// TIA Portal V20 export
FUNCTION "FNet_Map07" : Void   // FC143, LAD
// stored: Namespace CITI_Logic, SetENOAutomatically false
   VAR_TEMP
      FlexNet_DataString_PUN : Array[1..20] of Char;
      FlexNet_GM_PartNumber : Array[1..8] of Char;
      FlexNet_OptionalData : Array[1..12] of Char;
      FlexNet_Tracking_ID1 : Array[1..32] of Char;
      FlexNet_Track_ID1_Attrib : Array[1..20] of Char;
      FlexNet_Tracking_ID2 : Array[1..32] of Char;
      FlexNet_Track_ID2_Attrib : Array[1..20] of Char;
      FlexNet_Tracking_ID3 : Array[1..32] of Char;
      FlexNet_Track_ID3_Attrib : Array[1..20] of Char;
      FlexNet_Tracking_ID4 : Array[1..32] of Char;
      FlexNet_Track_ID4_Attrib : Array[1..20] of Char;
      FlexNet_Tracking_ID5 : Array[1..32] of Char;
      FlexNet_Track_ID5_Attrib : Array[1..20] of Char;
      FlexNet_Tracking_ID6 : Array[1..32] of Char;
      FlexNet_Track_ID6_Attrib : Array[1..20] of Char;
      FlexNet_Tracking_ID7 : Array[1..32] of Char;
      FlexNet_Track_ID7_Attrib : Array[1..20] of Char;
      FlexNet_Tracking_ID8 : Array[1..32] of Char;
      FlexNet_Track_ID8_Attrib : Array[1..20] of Char;
      FlexNet_Tracking_ID9 : Array[1..32] of Char;
      FlexNet_Track_ID9_Attrib : Array[1..20] of Char;
      FlexNet_Tracking_ID10 : Array[1..32] of Char;
      FlexNet_Track_ID10_Attrib : Array[1..20] of Char;
      TEMP_OEM_FnetNoRespWarn : Bool;   // REPLACE THIS WITH CORRECT WARNING BIT
      TEMP_OEM_FnetRetryOccur : Bool;   // REPLACE THIS WITH CORRECT WARNING BIT
      TEMP_OEM_FN_NoResponseL2 : Byte;
      OEM_FN_DATA_RECVD : Bool;
      TracePoint : Bool;
      Marriage : Bool;
      QualityGate : Bool;
      HostQuery : Bool;
      OEM_to_Populate_FN_RESPONSE_COUNTS_ALLOWED : Int;
   END_VAR
   VAR_TEMP   // added for the SCL form of the ladder/FBD networks
      _w1 : Bool;
      _w2 : Bool;
   END_VAR
BEGIN

REGION Network 1: Part Pass
   // **Replace the "CITI_Logic_Setup".OEM_TO_COMPLETE Bit with the correct Logic to drive the signal**
   // 
   // Set the Pass Bit Always True for a Trace Point, Marriage, and Host Query.
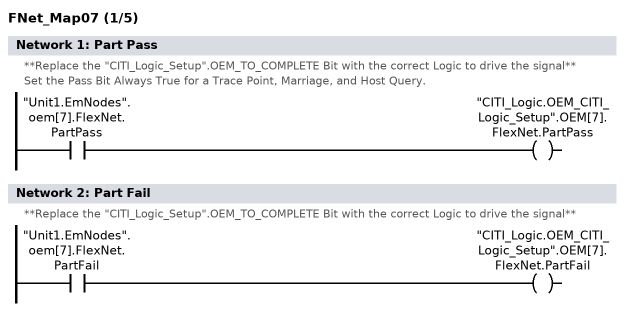
   RUNG wire#powerrail
      Contact( "Unit1.EmNodes".oem[7].FlexNet.PartPass )
      Coil( "CITI_Logic.OEM_CITI_Logic_Setup".OEM[7].FlexNet.PartPass )
   END_RUNG
   // the same network as SCL:
   "CITI_Logic.OEM_CITI_Logic_Setup".OEM[7].FlexNet.PartPass := "Unit1.EmNodes".oem[7].FlexNet.PartPass;
END_REGION

REGION Network 2: Part Fail
   // **Replace the "CITI_Logic_Setup".OEM_TO_COMPLETE Bit with the correct Logic to drive the signal**
   RUNG wire#powerrail
      Contact( "Unit1.EmNodes".oem[7].FlexNet.PartFail )
      Coil( "CITI_Logic.OEM_CITI_Logic_Setup".OEM[7].FlexNet.PartFail )
   END_RUNG
   // the same network as SCL:
   "CITI_Logic.OEM_CITI_Logic_Setup".OEM[7].FlexNet.PartFail := "Unit1.EmNodes".oem[7].FlexNet.PartFail;
END_REGION

REGION Network 3: Pun, GM Part Number, Optional Data, Tracking ID, Tracking ID Attribute, and Data Ready
   // **Replace the "CITI_Logic_Setup".OEM_TO_COMPLETE Bit with the correct Logic to drive the signal**
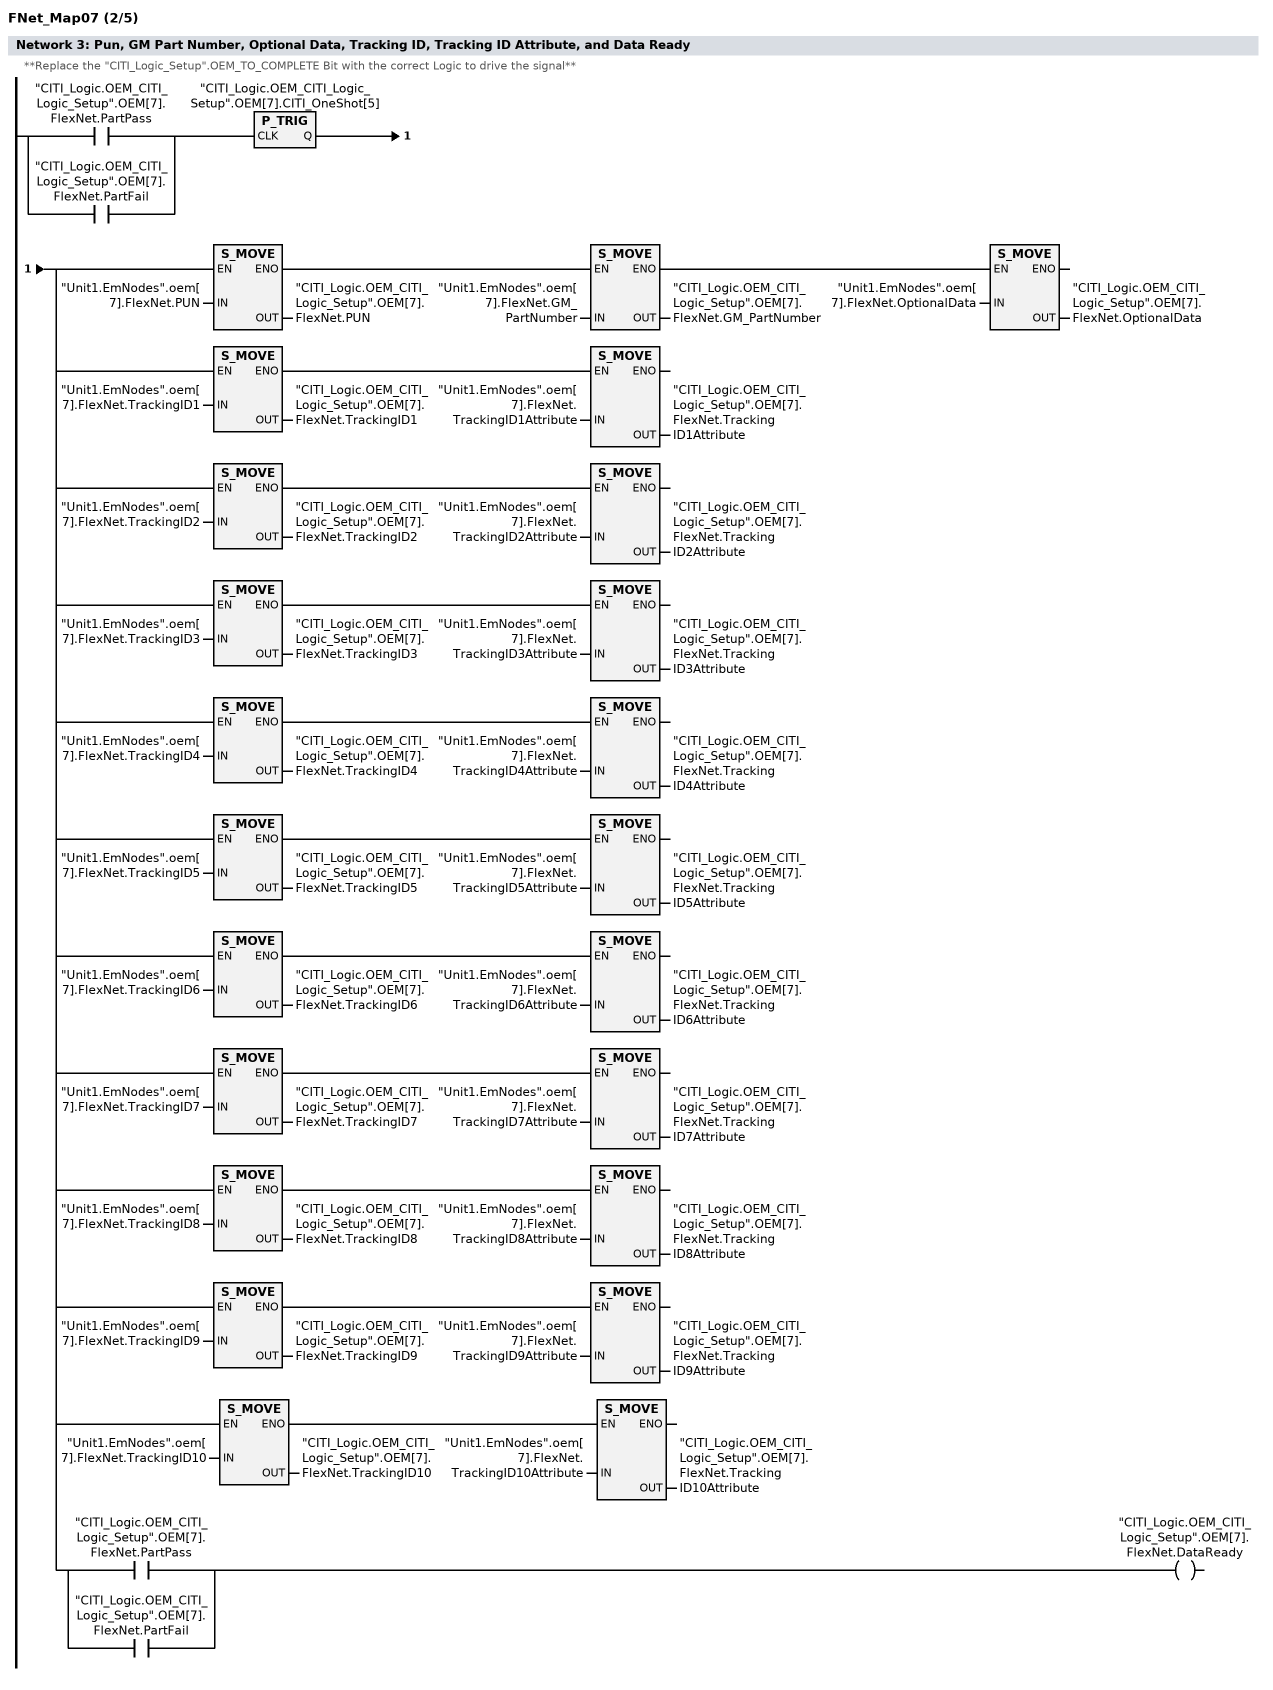
   RUNG wire#powerrail
      Contact( "CITI_Logic.OEM_CITI_Logic_Setup".OEM[7].FlexNet.PartPass )
      wire#w1
      P_Trig( "CITI_Logic.OEM_CITI_Logic_Setup".OEM[7].CITI_OneShot[5] )
      wire#w2
      S_Move(in := "Unit1.EmNodes".oem[7].FlexNet.PUN, out => "CITI_Logic.OEM_CITI_Logic_Setup".OEM[7].FlexNet.PUN)
      S_Move(in := "Unit1.EmNodes".oem[7].FlexNet.GM_PartNumber, out => "CITI_Logic.OEM_CITI_Logic_Setup".OEM[7].FlexNet.GM_PartNumber)
      S_Move(in := "Unit1.EmNodes".oem[7].FlexNet.OptionalData, out => "CITI_Logic.OEM_CITI_Logic_Setup".OEM[7].FlexNet.OptionalData)
   END_RUNG
   RUNG wire#powerrail
      Contact( "CITI_Logic.OEM_CITI_Logic_Setup".OEM[7].FlexNet.PartFail )
   END_RUNG wire#w1
   RUNG wire#w2
      S_Move(in := "Unit1.EmNodes".oem[7].FlexNet.TrackingID1, out => "CITI_Logic.OEM_CITI_Logic_Setup".OEM[7].FlexNet.TrackingID1)
      S_Move(in := "Unit1.EmNodes".oem[7].FlexNet.TrackingID1Attribute, out => "CITI_Logic.OEM_CITI_Logic_Setup".OEM[7].FlexNet.TrackingID1Attribute)
   END_RUNG
   RUNG wire#w2
      S_Move(in := "Unit1.EmNodes".oem[7].FlexNet.TrackingID2, out => "CITI_Logic.OEM_CITI_Logic_Setup".OEM[7].FlexNet.TrackingID2)
      S_Move(in := "Unit1.EmNodes".oem[7].FlexNet.TrackingID2Attribute, out => "CITI_Logic.OEM_CITI_Logic_Setup".OEM[7].FlexNet.TrackingID2Attribute)
   END_RUNG
   RUNG wire#w2
      S_Move(in := "Unit1.EmNodes".oem[7].FlexNet.TrackingID3, out => "CITI_Logic.OEM_CITI_Logic_Setup".OEM[7].FlexNet.TrackingID3)
      S_Move(in := "Unit1.EmNodes".oem[7].FlexNet.TrackingID3Attribute, out => "CITI_Logic.OEM_CITI_Logic_Setup".OEM[7].FlexNet.TrackingID3Attribute)
   END_RUNG
   RUNG wire#w2
      S_Move(in := "Unit1.EmNodes".oem[7].FlexNet.TrackingID4, out => "CITI_Logic.OEM_CITI_Logic_Setup".OEM[7].FlexNet.TrackingID4)
      S_Move(in := "Unit1.EmNodes".oem[7].FlexNet.TrackingID4Attribute, out => "CITI_Logic.OEM_CITI_Logic_Setup".OEM[7].FlexNet.TrackingID4Attribute)
   END_RUNG
   RUNG wire#w2
      S_Move(in := "Unit1.EmNodes".oem[7].FlexNet.TrackingID5, out => "CITI_Logic.OEM_CITI_Logic_Setup".OEM[7].FlexNet.TrackingID5)
      S_Move(in := "Unit1.EmNodes".oem[7].FlexNet.TrackingID5Attribute, out => "CITI_Logic.OEM_CITI_Logic_Setup".OEM[7].FlexNet.TrackingID5Attribute)
   END_RUNG
   RUNG wire#w2
      S_Move(in := "Unit1.EmNodes".oem[7].FlexNet.TrackingID6, out => "CITI_Logic.OEM_CITI_Logic_Setup".OEM[7].FlexNet.TrackingID6)
      S_Move(in := "Unit1.EmNodes".oem[7].FlexNet.TrackingID6Attribute, out => "CITI_Logic.OEM_CITI_Logic_Setup".OEM[7].FlexNet.TrackingID6Attribute)
   END_RUNG
   RUNG wire#w2
      S_Move(in := "Unit1.EmNodes".oem[7].FlexNet.TrackingID7, out => "CITI_Logic.OEM_CITI_Logic_Setup".OEM[7].FlexNet.TrackingID7)
      S_Move(in := "Unit1.EmNodes".oem[7].FlexNet.TrackingID7Attribute, out => "CITI_Logic.OEM_CITI_Logic_Setup".OEM[7].FlexNet.TrackingID7Attribute)
   END_RUNG
   RUNG wire#w2
      S_Move(in := "Unit1.EmNodes".oem[7].FlexNet.TrackingID8, out => "CITI_Logic.OEM_CITI_Logic_Setup".OEM[7].FlexNet.TrackingID8)
      S_Move(in := "Unit1.EmNodes".oem[7].FlexNet.TrackingID8Attribute, out => "CITI_Logic.OEM_CITI_Logic_Setup".OEM[7].FlexNet.TrackingID8Attribute)
   END_RUNG
   RUNG wire#w2
      S_Move(in := "Unit1.EmNodes".oem[7].FlexNet.TrackingID9, out => "CITI_Logic.OEM_CITI_Logic_Setup".OEM[7].FlexNet.TrackingID9)
      S_Move(in := "Unit1.EmNodes".oem[7].FlexNet.TrackingID9Attribute, out => "CITI_Logic.OEM_CITI_Logic_Setup".OEM[7].FlexNet.TrackingID9Attribute)
   END_RUNG
   RUNG wire#w2
      S_Move(in := "Unit1.EmNodes".oem[7].FlexNet.TrackingID10, out => "CITI_Logic.OEM_CITI_Logic_Setup".OEM[7].FlexNet.TrackingID10)
      S_Move(in := "Unit1.EmNodes".oem[7].FlexNet.TrackingID10Attribute, out => "CITI_Logic.OEM_CITI_Logic_Setup".OEM[7].FlexNet.TrackingID10Attribute)
   END_RUNG
   RUNG wire#w2
      Contact( "CITI_Logic.OEM_CITI_Logic_Setup".OEM[7].FlexNet.PartPass )
      wire#w3
      Coil( "CITI_Logic.OEM_CITI_Logic_Setup".OEM[7].FlexNet.DataReady )
   END_RUNG
   RUNG wire#w2
      Contact( "CITI_Logic.OEM_CITI_Logic_Setup".OEM[7].FlexNet.PartFail )
   END_RUNG wire#w3
   // the same network as SCL:
   #_w1 := "CITI_Logic.OEM_CITI_Logic_Setup".OEM[7].FlexNet.PartPass OR "CITI_Logic.OEM_CITI_Logic_Setup".OEM[7].FlexNet.PartFail;
   #_w2 := #_w1 AND NOT "CITI_Logic.OEM_CITI_Logic_Setup".OEM[7].CITI_OneShot[5];   // rising edge
   "CITI_Logic.OEM_CITI_Logic_Setup".OEM[7].CITI_OneShot[5] := #_w1;
   IF #_w2 THEN
       "CITI_Logic.OEM_CITI_Logic_Setup".OEM[7].FlexNet.PUN := "Unit1.EmNodes".oem[7].FlexNet.PUN;
       "CITI_Logic.OEM_CITI_Logic_Setup".OEM[7].FlexNet.GM_PartNumber := "Unit1.EmNodes".oem[7].FlexNet.GM_PartNumber;
       "CITI_Logic.OEM_CITI_Logic_Setup".OEM[7].FlexNet.OptionalData := "Unit1.EmNodes".oem[7].FlexNet.OptionalData;
       "CITI_Logic.OEM_CITI_Logic_Setup".OEM[7].FlexNet.TrackingID1 := "Unit1.EmNodes".oem[7].FlexNet.TrackingID1;
       "CITI_Logic.OEM_CITI_Logic_Setup".OEM[7].FlexNet.TrackingID1Attribute := "Unit1.EmNodes".oem[7].FlexNet.TrackingID1Attribute;
       "CITI_Logic.OEM_CITI_Logic_Setup".OEM[7].FlexNet.TrackingID2 := "Unit1.EmNodes".oem[7].FlexNet.TrackingID2;
       "CITI_Logic.OEM_CITI_Logic_Setup".OEM[7].FlexNet.TrackingID2Attribute := "Unit1.EmNodes".oem[7].FlexNet.TrackingID2Attribute;
       "CITI_Logic.OEM_CITI_Logic_Setup".OEM[7].FlexNet.TrackingID3 := "Unit1.EmNodes".oem[7].FlexNet.TrackingID3;
       "CITI_Logic.OEM_CITI_Logic_Setup".OEM[7].FlexNet.TrackingID3Attribute := "Unit1.EmNodes".oem[7].FlexNet.TrackingID3Attribute;
       "CITI_Logic.OEM_CITI_Logic_Setup".OEM[7].FlexNet.TrackingID4 := "Unit1.EmNodes".oem[7].FlexNet.TrackingID4;
       "CITI_Logic.OEM_CITI_Logic_Setup".OEM[7].FlexNet.TrackingID4Attribute := "Unit1.EmNodes".oem[7].FlexNet.TrackingID4Attribute;
       "CITI_Logic.OEM_CITI_Logic_Setup".OEM[7].FlexNet.TrackingID5 := "Unit1.EmNodes".oem[7].FlexNet.TrackingID5;
       "CITI_Logic.OEM_CITI_Logic_Setup".OEM[7].FlexNet.TrackingID5Attribute := "Unit1.EmNodes".oem[7].FlexNet.TrackingID5Attribute;
       "CITI_Logic.OEM_CITI_Logic_Setup".OEM[7].FlexNet.TrackingID6 := "Unit1.EmNodes".oem[7].FlexNet.TrackingID6;
       "CITI_Logic.OEM_CITI_Logic_Setup".OEM[7].FlexNet.TrackingID6Attribute := "Unit1.EmNodes".oem[7].FlexNet.TrackingID6Attribute;
       "CITI_Logic.OEM_CITI_Logic_Setup".OEM[7].FlexNet.TrackingID7 := "Unit1.EmNodes".oem[7].FlexNet.TrackingID7;
       "CITI_Logic.OEM_CITI_Logic_Setup".OEM[7].FlexNet.TrackingID7Attribute := "Unit1.EmNodes".oem[7].FlexNet.TrackingID7Attribute;
       "CITI_Logic.OEM_CITI_Logic_Setup".OEM[7].FlexNet.TrackingID8 := "Unit1.EmNodes".oem[7].FlexNet.TrackingID8;
       "CITI_Logic.OEM_CITI_Logic_Setup".OEM[7].FlexNet.TrackingID8Attribute := "Unit1.EmNodes".oem[7].FlexNet.TrackingID8Attribute;
       "CITI_Logic.OEM_CITI_Logic_Setup".OEM[7].FlexNet.TrackingID9 := "Unit1.EmNodes".oem[7].FlexNet.TrackingID9;
       "CITI_Logic.OEM_CITI_Logic_Setup".OEM[7].FlexNet.TrackingID9Attribute := "Unit1.EmNodes".oem[7].FlexNet.TrackingID9Attribute;
       "CITI_Logic.OEM_CITI_Logic_Setup".OEM[7].FlexNet.TrackingID10 := "Unit1.EmNodes".oem[7].FlexNet.TrackingID10;
       "CITI_Logic.OEM_CITI_Logic_Setup".OEM[7].FlexNet.TrackingID10Attribute := "Unit1.EmNodes".oem[7].FlexNet.TrackingID10Attribute;
   END_IF;
   "CITI_Logic.OEM_CITI_Logic_Setup".OEM[7].FlexNet.DataReady := #_w2 AND ("CITI_Logic.OEM_CITI_Logic_Setup".OEM[7].FlexNet.PartPass OR "CITI_Logic.OEM_CITI_Logic_Setup".OEM[7].FlexNet.PartFail);
END_REGION

REGION Network 4: Transaction Type
   // **Replace the "CITI_Logic_Setup".OEM_TO_COMPLETE Bit with the correct Logic to drive the signal**
   // 
   // For the Transaction Type:
   //  
   // Flexnet TypeInteger Value
   // Trace Point = 1
   // Marriage = 2
   // Quality Gate = 4
   // Host Query = 8
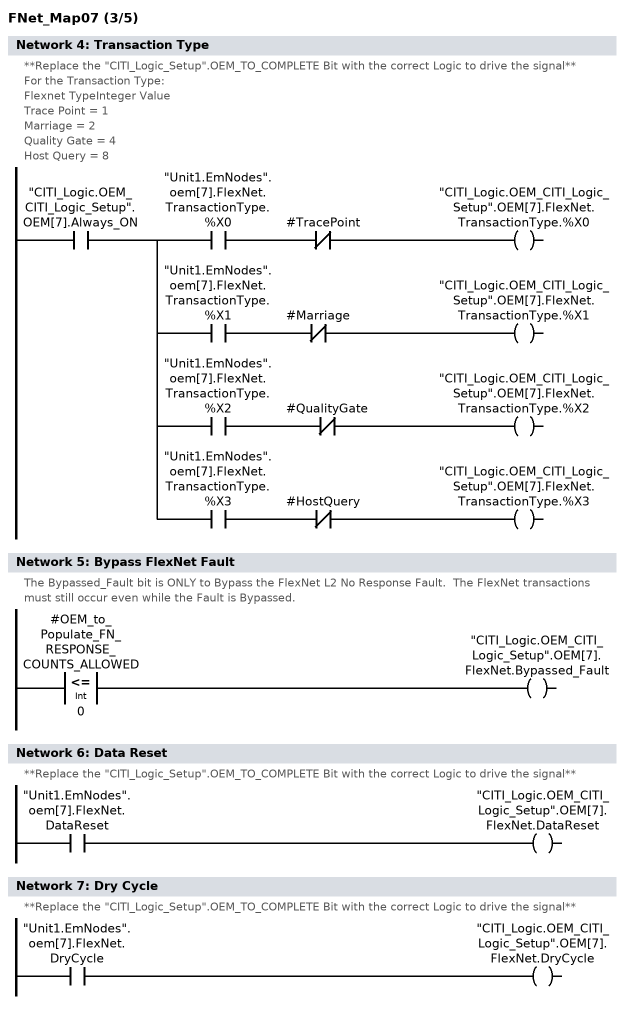
   RUNG wire#powerrail
      Contact( "CITI_Logic.OEM_CITI_Logic_Setup".OEM[7].Always_ON )
      wire#w1
      Contact( "Unit1.EmNodes".oem[7].FlexNet.TransactionType.%X0 )
      I_Contact( #TracePoint )
      Coil( "CITI_Logic.OEM_CITI_Logic_Setup".OEM[7].FlexNet.TransactionType.%X0 )
   END_RUNG
   RUNG wire#w1
      Contact( "Unit1.EmNodes".oem[7].FlexNet.TransactionType.%X1 )
      I_Contact( #Marriage )
      Coil( "CITI_Logic.OEM_CITI_Logic_Setup".OEM[7].FlexNet.TransactionType.%X1 )
   END_RUNG
   RUNG wire#w1
      Contact( "Unit1.EmNodes".oem[7].FlexNet.TransactionType.%X2 )
      I_Contact( #QualityGate )
      Coil( "CITI_Logic.OEM_CITI_Logic_Setup".OEM[7].FlexNet.TransactionType.%X2 )
   END_RUNG
   RUNG wire#w1
      Contact( "Unit1.EmNodes".oem[7].FlexNet.TransactionType.%X3 )
      I_Contact( #HostQuery )
      Coil( "CITI_Logic.OEM_CITI_Logic_Setup".OEM[7].FlexNet.TransactionType.%X3 )
   END_RUNG
   // the same network as SCL:
   #_w1 := "CITI_Logic.OEM_CITI_Logic_Setup".OEM[7].Always_ON;
   "CITI_Logic.OEM_CITI_Logic_Setup".OEM[7].FlexNet.TransactionType.%X0 := "CITI_Logic.OEM_CITI_Logic_Setup".OEM[7].Always_ON AND "Unit1.EmNodes".oem[7].FlexNet.TransactionType.%X0 AND NOT #TracePoint;
   "CITI_Logic.OEM_CITI_Logic_Setup".OEM[7].FlexNet.TransactionType.%X1 := #_w1 AND "Unit1.EmNodes".oem[7].FlexNet.TransactionType.%X1 AND NOT #Marriage;
   "CITI_Logic.OEM_CITI_Logic_Setup".OEM[7].FlexNet.TransactionType.%X2 := #_w1 AND "Unit1.EmNodes".oem[7].FlexNet.TransactionType.%X2 AND NOT #QualityGate;
   "CITI_Logic.OEM_CITI_Logic_Setup".OEM[7].FlexNet.TransactionType.%X3 := #_w1 AND "Unit1.EmNodes".oem[7].FlexNet.TransactionType.%X3 AND NOT #HostQuery;
END_REGION

REGION Network 5: Bypass FlexNet Fault
   // The Bypassed_Fault bit is ONLY to Bypass the FlexNet L2 No Response Fault.  The FlexNet transactions must still occur even while the Fault is Bypassed.
   RUNG wire#powerrail
      { S7_Templates := "SrcType := Int" } LE_Contact(in1 := #OEM_to_Populate_FN_RESPONSE_COUNTS_ALLOWED, in2 := 0)
      Coil( "CITI_Logic.OEM_CITI_Logic_Setup".OEM[7].FlexNet.Bypassed_Fault )
   END_RUNG
   // the same network as SCL:
   "CITI_Logic.OEM_CITI_Logic_Setup".OEM[7].FlexNet.Bypassed_Fault := #OEM_to_Populate_FN_RESPONSE_COUNTS_ALLOWED <= 0;
END_REGION

REGION Network 6: Data Reset
   // **Replace the "CITI_Logic_Setup".OEM_TO_COMPLETE Bit with the correct Logic to drive the signal**
   RUNG wire#powerrail
      Contact( "Unit1.EmNodes".oem[7].FlexNet.DataReset )
      Coil( "CITI_Logic.OEM_CITI_Logic_Setup".OEM[7].FlexNet.DataReset )
   END_RUNG
   // the same network as SCL:
   "CITI_Logic.OEM_CITI_Logic_Setup".OEM[7].FlexNet.DataReset := "Unit1.EmNodes".oem[7].FlexNet.DataReset;
END_REGION

REGION Network 7: Dry Cycle
   // **Replace the "CITI_Logic_Setup".OEM_TO_COMPLETE Bit with the correct Logic to drive the signal**
   RUNG wire#powerrail
      Contact( "Unit1.EmNodes".oem[7].FlexNet.DryCycle )
      Coil( "CITI_Logic.OEM_CITI_Logic_Setup".OEM[7].FlexNet.DryCycle )
   END_RUNG
   // the same network as SCL:
   "CITI_Logic.OEM_CITI_Logic_Setup".OEM[7].FlexNet.DryCycle := "Unit1.EmNodes".oem[7].FlexNet.DryCycle;
END_REGION

REGION Network 8: FlexNet 10 Child Block Call
   // Input time for response fault can be directly entered or from another source.
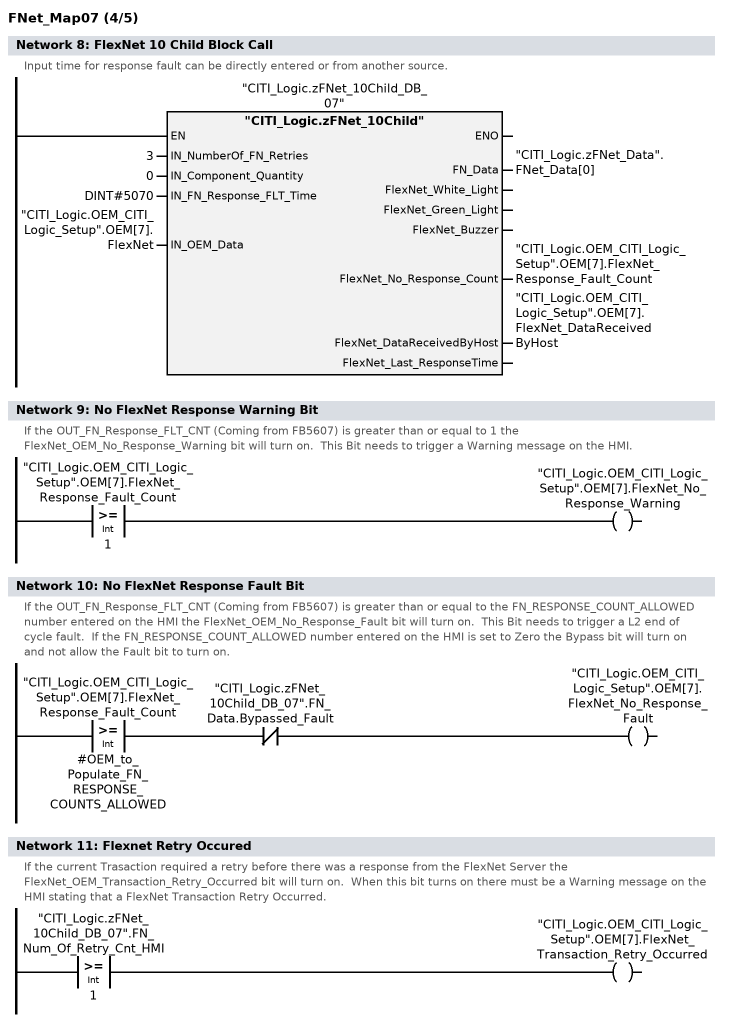
   RUNG wire#powerrail
      "CITI_Logic.zFNet_10Child_DB_07"(IN_NumberOf_FN_Retries := 3, IN_Component_Quantity := 0, IN_FN_Response_FLT_Time := DINT#5070, IN_OEM_Data := "CITI_Logic.OEM_CITI_Logic_Setup".OEM[7].FlexNet, FN_Data => "CITI_Logic.zFNet_Data".FNet_Data[0], FlexNet_White_Light =>, FlexNet_Green_Light =>, FlexNet_Buzzer =>, FlexNet_No_Response_Count => "CITI_Logic.OEM_CITI_Logic_Setup".OEM[7].FlexNet_Response_Fault_Count, FlexNet_DataReceivedByHost => "CITI_Logic.OEM_CITI_Logic_Setup".OEM[7].FlexNet_DataReceivedByHost, FlexNet_Last_ResponseTime =>)
   END_RUNG
   // the same network as SCL:
   "CITI_Logic.zFNet_10Child_DB_07"(IN_NumberOf_FN_Retries := 3,   // "CITI_Logic.zFNet_10Child"
                           IN_Component_Quantity := 0,
                           IN_FN_Response_FLT_Time := DINT#5070,
                           IN_OEM_Data := "CITI_Logic.OEM_CITI_Logic_Setup".OEM[7].FlexNet,
                           FN_Data => "CITI_Logic.zFNet_Data".FNet_Data[0],
                           FlexNet_No_Response_Count => "CITI_Logic.OEM_CITI_Logic_Setup".OEM[7].FlexNet_Response_Fault_Count,
                           FlexNet_DataReceivedByHost => "CITI_Logic.OEM_CITI_Logic_Setup".OEM[7].FlexNet_DataReceivedByHost);
END_REGION

REGION Network 9: No FlexNet Response Warning Bit
   // If the OUT_FN_Response_FLT_CNT (Coming from FB5607) is greater than or equal to 1 the FlexNet_OEM_No_Response_Warning bit will turn on.  This Bit needs to trigger a Warning message on the HMI.
   RUNG wire#powerrail
      { S7_Templates := "SrcType := Int" } GE_Contact(in1 := "CITI_Logic.OEM_CITI_Logic_Setup".OEM[7].FlexNet_Response_Fault_Count, in2 := 1)
      Coil( "CITI_Logic.OEM_CITI_Logic_Setup".OEM[7].FlexNet_No_Response_Warning )
   END_RUNG
   // the same network as SCL:
   "CITI_Logic.OEM_CITI_Logic_Setup".OEM[7].FlexNet_No_Response_Warning := "CITI_Logic.OEM_CITI_Logic_Setup".OEM[7].FlexNet_Response_Fault_Count >= 1;
END_REGION

REGION Network 10: No FlexNet Response Fault Bit
   // If the OUT_FN_Response_FLT_CNT (Coming from FB5607) is greater than or equal to the FN_RESPONSE_COUNT_ALLOWED number entered on the HMI the FlexNet_OEM_No_Response_Fault bit will turn on.  This Bit needs to trigger a L2 end of cycle fault.  If the FN_RESPONSE_COUNT_ALLOWED number entered on the HMI is set to Zero the Bypass bit will turn on and not allow the Fault bit to turn on.
   RUNG wire#powerrail
      { S7_Templates := "SrcType := Int" } GE_Contact(in1 := "CITI_Logic.OEM_CITI_Logic_Setup".OEM[7].FlexNet_Response_Fault_Count, in2 := #OEM_to_Populate_FN_RESPONSE_COUNTS_ALLOWED)
      I_Contact( "CITI_Logic.zFNet_10Child_DB_07".FN_Data.Bypassed_Fault )
      Coil( "CITI_Logic.OEM_CITI_Logic_Setup".OEM[7].FlexNet_No_Response_Fault )
   END_RUNG
   // the same network as SCL:
   "CITI_Logic.OEM_CITI_Logic_Setup".OEM[7].FlexNet_No_Response_Fault := ("CITI_Logic.OEM_CITI_Logic_Setup".OEM[7].FlexNet_Response_Fault_Count >= #OEM_to_Populate_FN_RESPONSE_COUNTS_ALLOWED) AND NOT "CITI_Logic.zFNet_10Child_DB_07".FN_Data.Bypassed_Fault;
END_REGION

REGION Network 11: Flexnet Retry Occured
   // If the current Trasaction required a retry before there was a response from the FlexNet Server the FlexNet_OEM_Transaction_Retry_Occurred bit will turn on.  When this bit turns on there must be a Warning message on the HMI stating that a FlexNet Transaction Retry Occurred.
   RUNG wire#powerrail
      { S7_Templates := "SrcType := Int" } GE_Contact(in1 := "CITI_Logic.zFNet_10Child_DB_07".FN_Num_Of_Retry_Cnt_HMI, in2 := 1)
      Coil( "CITI_Logic.OEM_CITI_Logic_Setup".OEM[7].FlexNet_Transaction_Retry_Occurred )
   END_RUNG
   // the same network as SCL:
   "CITI_Logic.OEM_CITI_Logic_Setup".OEM[7].FlexNet_Transaction_Retry_Occurred := "CITI_Logic.zFNet_10Child_DB_07".FN_Num_Of_Retry_Cnt_HMI >= 1;
END_REGION

REGION Network 12: FlexNet Host Query "Part NOK" Example Fault for Machining
   // This example shows how to structure the responses for the Parent Part Good/Hold and a couple of the Tracking Components Good/Hold.  Please add additional tracking components if they are used or delete any tracking components that are not needed.
   // 
   // This is an example. The OEM is responsible for the correct implementation.
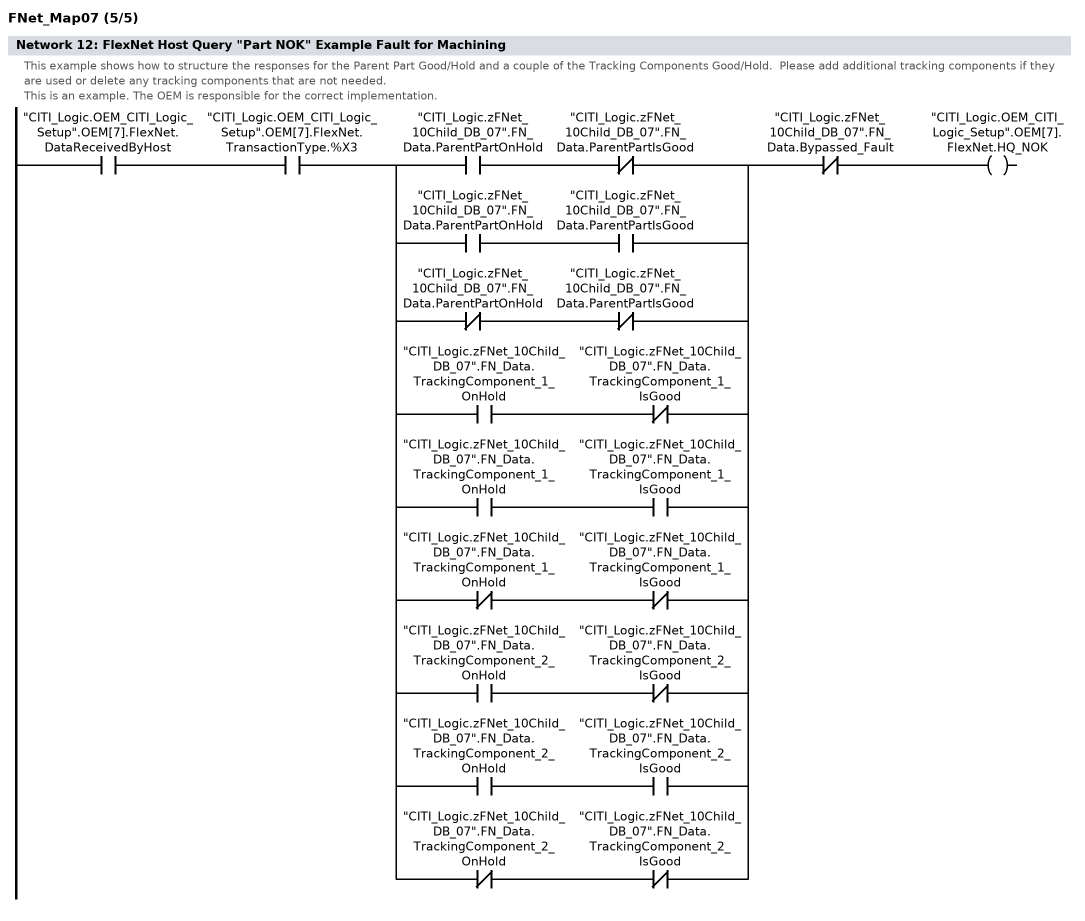
   RUNG wire#powerrail
      Contact( "CITI_Logic.OEM_CITI_Logic_Setup".OEM[7].FlexNet.DataReceivedByHost )
      Contact( "CITI_Logic.OEM_CITI_Logic_Setup".OEM[7].FlexNet.TransactionType.%X3 )
      wire#w1
      Contact( "CITI_Logic.zFNet_10Child_DB_07".FN_Data.ParentPartOnHold )
      I_Contact( "CITI_Logic.zFNet_10Child_DB_07".FN_Data.ParentPartIsGood )
      wire#w2
      I_Contact( "CITI_Logic.zFNet_10Child_DB_07".FN_Data.Bypassed_Fault )
      Coil( "CITI_Logic.OEM_CITI_Logic_Setup".OEM[7].FlexNet.HQ_NOK )
   END_RUNG
   RUNG wire#w1
      Contact( "CITI_Logic.zFNet_10Child_DB_07".FN_Data.ParentPartOnHold )
      Contact( "CITI_Logic.zFNet_10Child_DB_07".FN_Data.ParentPartIsGood )
   END_RUNG wire#w2
   RUNG wire#w1
      I_Contact( "CITI_Logic.zFNet_10Child_DB_07".FN_Data.ParentPartOnHold )
      I_Contact( "CITI_Logic.zFNet_10Child_DB_07".FN_Data.ParentPartIsGood )
   END_RUNG wire#w2
   RUNG wire#w1
      Contact( "CITI_Logic.zFNet_10Child_DB_07".FN_Data.TrackingComponent_1_OnHold )
      I_Contact( "CITI_Logic.zFNet_10Child_DB_07".FN_Data.TrackingComponent_1_IsGood )
   END_RUNG wire#w2
   RUNG wire#w1
      Contact( "CITI_Logic.zFNet_10Child_DB_07".FN_Data.TrackingComponent_1_OnHold )
      Contact( "CITI_Logic.zFNet_10Child_DB_07".FN_Data.TrackingComponent_1_IsGood )
   END_RUNG wire#w2
   RUNG wire#w1
      I_Contact( "CITI_Logic.zFNet_10Child_DB_07".FN_Data.TrackingComponent_1_OnHold )
      I_Contact( "CITI_Logic.zFNet_10Child_DB_07".FN_Data.TrackingComponent_1_IsGood )
   END_RUNG wire#w2
   RUNG wire#w1
      Contact( "CITI_Logic.zFNet_10Child_DB_07".FN_Data.TrackingComponent_2_OnHold )
      I_Contact( "CITI_Logic.zFNet_10Child_DB_07".FN_Data.TrackingComponent_2_IsGood )
   END_RUNG wire#w2
   RUNG wire#w1
      Contact( "CITI_Logic.zFNet_10Child_DB_07".FN_Data.TrackingComponent_2_OnHold )
      Contact( "CITI_Logic.zFNet_10Child_DB_07".FN_Data.TrackingComponent_2_IsGood )
   END_RUNG wire#w2
   RUNG wire#w1
      I_Contact( "CITI_Logic.zFNet_10Child_DB_07".FN_Data.TrackingComponent_2_OnHold )
      I_Contact( "CITI_Logic.zFNet_10Child_DB_07".FN_Data.TrackingComponent_2_IsGood )
   END_RUNG wire#w2
   // the same network as SCL:
   "CITI_Logic.OEM_CITI_Logic_Setup".OEM[7].FlexNet.HQ_NOK := "CITI_Logic.OEM_CITI_Logic_Setup".OEM[7].FlexNet.DataReceivedByHost AND "CITI_Logic.OEM_CITI_Logic_Setup".OEM[7].FlexNet.TransactionType.%X3 AND (("CITI_Logic.zFNet_10Child_DB_07".FN_Data.ParentPartOnHold AND NOT "CITI_Logic.zFNet_10Child_DB_07".FN_Data.ParentPartIsGood) OR ("CITI_Logic.zFNet_10Child_DB_07".FN_Data.ParentPartOnHold AND "CITI_Logic.zFNet_10Child_DB_07".FN_Data.ParentPartIsGood) OR (NOT "CITI_Logic.zFNet_10Child_DB_07".FN_Data.ParentPartOnHold AND NOT "CITI_Logic.zFNet_10Child_DB_07".FN_Data.ParentPartIsGood) OR ("CITI_Logic.zFNet_10Child_DB_07".FN_Data.TrackingComponent_1_OnHold AND NOT "CITI_Logic.zFNet_10Child_DB_07".FN_Data.TrackingComponent_1_IsGood) OR ("CITI_Logic.zFNet_10Child_DB_07".FN_Data.TrackingComponent_1_OnHold AND "CITI_Logic.zFNet_10Child_DB_07".FN_Data.TrackingComponent_1_IsGood) OR (NOT "CITI_Logic.zFNet_10Child_DB_07".FN_Data.TrackingComponent_1_OnHold AND NOT "CITI_Logic.zFNet_10Child_DB_07".FN_Data.TrackingComponent_1_IsGood) OR ("CITI_Logic.zFNet_10Child_DB_07".FN_Data.TrackingComponent_2_OnHold AND NOT "CITI_Logic.zFNet_10Child_DB_07".FN_Data.TrackingComponent_2_IsGood) OR ("CITI_Logic.zFNet_10Child_DB_07".FN_Data.TrackingComponent_2_OnHold AND "CITI_Logic.zFNet_10Child_DB_07".FN_Data.TrackingComponent_2_IsGood) OR (NOT "CITI_Logic.zFNet_10Child_DB_07".FN_Data.TrackingComponent_2_OnHold AND NOT "CITI_Logic.zFNet_10Child_DB_07".FN_Data.TrackingComponent_2_IsGood)) AND NOT "CITI_Logic.zFNet_10Child_DB_07".FN_Data.Bypassed_Fault;
END_REGION
END_FUNCTION
